// TIA Portal V20 export
VAR_GLOBAL   // PLC tag table "Standard-Variablentabelle"
   test0ibn AT %M0.4 : Bool;
   test1ibn AT %M0.5 : Bool;
   Tag_1 AT %M400.0 : Bool;
   Tag_2 AT %M400.1 : Bool;
   Tag_3 AT %M400.2 : Bool;
   Tag_4 AT %M2345.4 : Bool;
END_VAR
VAR_GLOBAL CONSTANT   // user constants
   USERDIAG_DEVICES_PER_SCREEN_UPPER_LIM : Int := 32;
   USERDIAG_SLOTS_PER_SCREEN_UPPER_LIM : Int := 31;
   USERDIAG_SLOTS_PER_DEVICE_UPPER_LIM : Int := 31;
   USERDIAG_DEVICES_PER_IO_SYSTEM_UPPER_LIM : Int := 128;
   USERDIAG_SLOTS_PER_PLC_UPPER_LIM : Int := 31;
END_VAR
